// Abstract class/Function Block that all collections inherit.
// Contains inheritable helper methods and base implementation
// for methods and properties for creating a collection.
{attribute 'enable_dynamic_creation'}
{attribute 'no_explicit_call' := 'direct call for this function block is not allowed'}
FUNCTION_BLOCK ABSTRACT FB_Collection IMPLEMENTS I_Collection
VAR
	Count : T_Capacity;
	Error : T_Error := (bStatus := FALSE, nCode := GVL_Errors.ERR_OK, sSource := 'No Error.');
END_VAR

// Number of items in the collection.
PROPERTY _Count : T_Capacity
GET
_Count := THIS^.Count;
END_GET
SET // PROTECTED
THIS^.Count := _Count;
END_SET
END_PROPERTY

// Checks if collection is empty.
PROPERTY _Empty : BOOL
GET
_Empty := THIS^._Count <= 0;
END_GET
END_PROPERTY

// Error status of the collection.
PROPERTY _Error_Status : T_Error
GET
_Error_Status := THIS^.Error;
END_GET
SET // PROTECTED
THIS^.Error := _Error_Status;
END_SET
END_PROPERTY

METHOD PROTECTED Clear_Error
VAR_INPUT
END_VAR
THIS^._Error_Status := F_Error(0,0,'');
END_METHOD

// Decrement collection count by 1.
METHOD PROTECTED Decrement_Count
THIS^._Count := THIS^._Count - 1;
END_METHOD

// Increments collection count by 1
METHOD PROTECTED Increment_Count
VAR_INPUT
END_VAR
THIS^._Count := THIS^._Count + 1;
END_METHOD

END_FUNCTION_BLOCK

(* stored: Version 1.1.0.1, ProductVersion 3.1.4024.4
   POU FB_Collection: Id {7742cad6-cf07-0c6e-381d-54d92eee7230}, SpecialFunc None
   Folder Protected: Id {dafbf2f8-a1aa-0dc3-14ad-1bab7f8f36e0}
   Property _Count: Id {26b379f5-40ad-064d-3faf-8e917bdfeaae}
   Get Get: Id {e0894d02-2319-02b4-2f05-03704cc729c7}
   Set Set: Id {439d8e64-6861-058a-2f58-0d1132366a2d}
   Property _Empty: Id {8290ebb5-2a66-0ab9-2091-8f592a26cca5}
   Get Get: Id {9e16e4fb-101a-0896-080b-b086925cabcd}
   Property _Error_Status: Id {b13cb86a-4979-07d5-22fe-e75f85a83eee}
   Get Get: Id {29540553-64a1-0f89-3626-ede965f403f3}
   Set Set: Id {13c9a81c-bd7d-05cb-006b-9f5168f136d7}
   Method Clear_Error: Id {56214d32-03a5-05b7-267e-3a7bf0140f9b}
   Method Decrement_Count: Id {6870a1c1-1f8d-035b-002e-86525d99ae88}
   Method Increment_Count: Id {b1768fd9-4b59-029a-30b3-52d595ca45fd} *)
